(* CoDeSys 2.3.9.62 project: main.pro *)
(* Libraries: Standard.lib, Iecsfc.lib 8.11.10 11:37:48, SYSLIBCALLBACK.LIB *)

(* PLC configuration (modules and I/O channels)
K-Bus [K_Bus] node 0, in %IB0 out %QB0
Internal Digital I/O [InternalDigIO] node 1, in %IB512 out %QB512
  Internal Digital Inputs [Internal_DIN] node 0, in %IB512 out %QB512
    DIN1 AT %IX2300.0 [BOOLOnX_I] Internal Digital Input Bit 1
    DIN2 AT %IX2300.1 [BOOLOnX_I] Internal Digital Input Bit 2
  Internal Digital Outputs [Internal_DOUT] node 1, in %IB513 out %QB512
    DOUT1 AT %QX2300.0 [BOOLOnX_Q] Internal Digital Output Bit 1
    DOUT2 AT %QX2300.1 [BOOLOnX_Q] Internal Digital Output Bit 2
Fieldbus variables [FB_VARS] node 3, in %IB0 out %QB0
Flag variables [FLAG_VARS] node 4, in %IB0 out %QB0
Modbus-Master [MB_MASTER] node 5, in %IB0 out %QB0
*)

(* Task configuration *)
TASK RunMainProgram (PRIORITY := 15);
	main();
END_TASK

(* POU main, ST *)
PROGRAM main
VAR
	counter : INT;
END_VAR
counter := counter + 1;

counter := counter + counter;
END_PROGRAM
